TYPE FB_ServoAchse_Hand :
STRUCT
	//Verfahren in positive Richtung
	pos : BOOL;
	//Verfahren in negative Richtung
	neg : BOOL;
END_STRUCT
END_TYPE

(* stored: Version 1.1.0.1, ProductVersion 3.1.4018.5
   DUT FB_ServoAchse_Hand: Id {813c13a1-e098-49f0-b10d-4d85669df82f} *)
